ABB RobotStudio station: Solution2_20190821-011730.rsstn

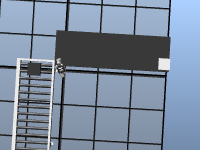
Station Solution2 (saved by RobotStudio 7.0.8504.151)
Controller Vinnie, task T_ROB1: task frame (RAPID world) sits at (0, 0, 400) mm in the station
Controller Vinnie
  mechanical unit ROB_1: IRB120_3_58__01, 6 joints, base frame (0, 0, 0) mm
Layout (positions relative to the parent item):
  - IRB120_3_58__01 [mechanism, from Robots\IRB120_3_58_G_01.rslib] at (0, 0, 400) mm; joint values [0.3488, 0.4268, 0.7489, 0, 0.3951, 0.3488] (rad or m)
  - Conveyor1 [smart component]
      signals: DI NewBox, DO BoxAtPos
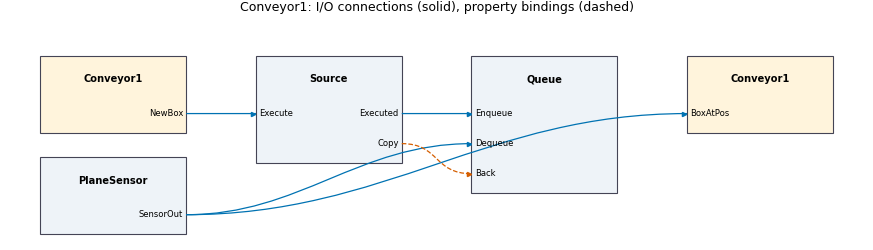
      connections:
        Conveyor1.NewBox -> Source.Execute
        Source.Executed -> Queue.Enqueue
        PlaneSensor.SensorOut -> Queue.Dequeue
        PlaneSensor.SensorOut -> Conveyor1.BoxAtPos
        Source.Copy => Queue.Back
    - 950_4000_h2 [part, from Equipment\Conveyor 950 4000 h2.rslib] at (-3846.63, 300, 0) mm
    - Source [smart component, from Components\Source.rslib]
        properties: Source=Part_1; Copy=Part_1_9; Parent=(none); Position=[0 0 0]; Orientation=[0 0 0]; Transient=false; PhysicsBehavior=0
    - Queue [smart component, from Components\Queue.rslib]
        properties: Back=Part_1_9; Front=(none); Queue={2cd56b75-4092-4768-a475-00f35c4dae8b};{e0dd32b4-5c51-4f0d-a48d-accb6fe5d5c2};{74c91f28-67c0-4405-bb46-46a2bebc9ae4};{4de452c9-d932-4406-abf8-51a8521f936e};{88fa9637-5f31-4297-a4ce-dfd895462f0a};{a1be2565-d57b-44ca-a3d4-488ed4227e35};{48cd2ff7-af39-436b-9b86-b527ae4f2f15};{69c433ef-7d00-473a-887e-093ac5fd6830}; NumberOfObjects=0
    - LinearMover [smart component, from Components\LinearMover.rslib]
        properties: Object=Queue; Direction=[1 0 0]; Speed=0.5; Reference=Global; ReferenceObject=(none)
    - PlaneSensor [smart component, from Components\PlaneSensor.rslib]
        properties: Origin=[0.162459 1.21 0.435]; Axis1=[0 -0.91 0]; Axis2=[0 0 0.2]; SensedPart=Part_1_9
      - _sensorPart_ [part]
  - Part_1 [part]
  - Part_1_9 [part] at (3480, 0, 0) mm
  - Conveyor2 [smart component]
    - Part_3 [part]
    - Source [smart component, from Components\Source.rslib]
        properties: Source=Part_4; Copy=(none); Parent=(none); Position=[0 0 0]; Orientation=[0 0 0]; Transient=false; PhysicsBehavior=0
    - LinearMover [smart component, from Components\LinearMover.rslib]
        properties: Object=Queue; Direction=[0 1 0]; Speed=0.5; Reference=Global; ReferenceObject=(none)
    - Queue [smart component, from Components\Queue.rslib]
        properties: Back=(none); Front=(none); Queue=; NumberOfObjects=0
    - PlaneSensor [smart component, from Components\PlaneSensor.rslib]
        properties: Origin=[0 0 0]; Axis1=[0.1 0 0]; Axis2=[0 0.1 0]; SensedPart=(none)
      - _sensorPart_ [part, from Components\PlaneSensor.rslib]
  - Part_4 [part]
